Omron CX-Programmer project NewProject (CX-Programmer 9.54)

# PLC program2: CJ1M CPU11

## Global symbols (name address type ; comment)
0.01 BOOL  ; startpb
0.02 BOOL  ; stoppb
0.03 BOOL  ; drillup
0.04 BOOL  ; drilldown
100.00 BOOL  ; forward rotating mot
100.01 BOOL  ; reverse rotating
10.00 BOOL  ; mem1

## Program NewProgram1 (cyclic task 0)

### Section Section1

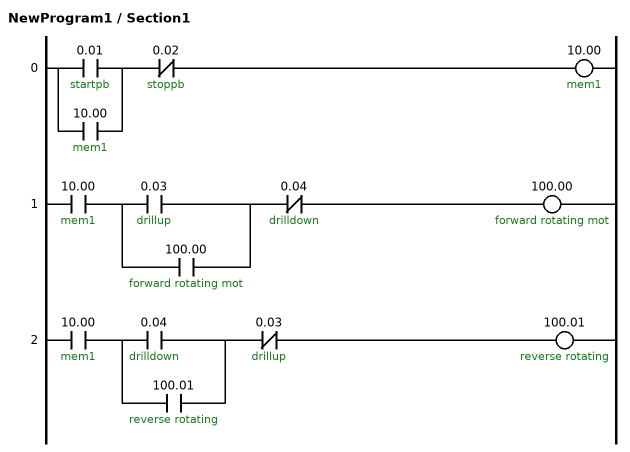
; rung 0
LD 0.01  ; startpb
OR 10.00  ; mem1
ANDNOT 0.02  ; stoppb
OUT 10.00  ; mem1
; rung 1
LD 10.00  ; mem1
LD 0.03  ; drillup
OR 100.00  ; forward rotating mot
ANDLD
ANDNOT 0.04  ; drilldown
OUT 100.00  ; forward rotating mot
; rung 2
LD 10.00  ; mem1
LD 0.04  ; drilldown
OR 100.01  ; reverse rotating
ANDLD
ANDNOT 0.03  ; drillup
OUT 100.01  ; reverse rotating

### Section END
; rung 0
END(001)